FUNCTION_BLOCK Q_ExecuteExtendedMacro (* Command Execute Extended Macro( Part 6 - F.62 ) *)
  (* Standard: ISO 11783-6; Description: This command is used to execute a Macro with 16-bit Object ID. This message is available in VT version 5 and later. Return values iso_s16 - E_NO_ERR - OK - E_OVERFLOW - buffer overflow - E_NOACT - Command not possible in current state - E_NO_INSTANCE - No VT client available *)
  (* Version 1.0, 2022-07-08, franz *)
  (* Documentation:
  This command is used to execute a Macro with 16-bit Object ID. This message is available in VT version 5 and later.
   Return values
   iso_s16
    - E_NO_ERR - OK
   - E_OVERFLOW - buffer overflow
   - E_NOACT - Command not possible in current state
   - E_NO_INSTANCE - No VT client available
  *)
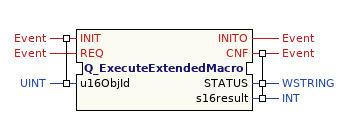
  EVENT_INPUT
    INIT WITH u16ObjId; (* Service Initialization *)
    REQ; (* Service Request *)
  END_EVENT
  EVENT_OUTPUT
    INITO; (* Initialization Confirm *)
    CNF WITH STATUS, s16result; (* Confirmation of Requested Service *)
  END_EVENT
  VAR_INPUT
    u16ObjId : UINT; (* Object ID of Macro object *)
  END_VAR
  VAR_OUTPUT
    STATUS : WSTRING; (* Service Status *)
    s16result : INT; (* retval see description *)
  END_VAR
END_FUNCTION_BLOCK
